{attribute 'linkalways'} 
{attribute 'no_explicit_call' := 'This FB is a CLASS and must be accessed using methods or properties'}
{attribute 'enable_dynamic_creation'}
FUNCTION_BLOCK AsynchronousRpcHandlers IMPLEMENTS I_AsynchronousRpcHandlers, I_HostAsynchronousRpcHandlers
VAR
	handlers : Dictionary;
	_hasHandlers : BOOL;
END_VAR

PROPERTY PUBLIC HasHandlers : BOOL
GET
HasHandlers := _hasHandlers;
END_GET
END_PROPERTY

METHOD PUBLIC RegisterHandler
VAR_INPUT
	MethodName : T_MAXSTRING;
	Handler : I_AsynchronousRpcHandler;
END_VAR
handlers.AddOrUpdate(MethodName, Handler);
_hasHandlers := true;
END_METHOD

METHOD PUBLIC TryGetByMethodName : BOOL
VAR_INPUT
	MethodName : T_MAXSTRING;
	Destination : REFERENCE TO I_AsynchronousRpcHandler;
END_VAR
TryGetByMethodName := handlers.TryGetValue(MethodName, Destination);
END_METHOD

END_FUNCTION_BLOCK

(* stored: Version 1.1.0.1, ProductVersion 3.1.4024.12
   POU AsynchronousRpcHandlers: Id {cd13ebd0-3788-4442-8ef7-64929a08abe4}, SpecialFunc None
   Property HasHandlers: Id {17926476-6420-47b5-979d-bcd741790e01}
   Get Get: Id {68a58ba0-9e12-4a74-b13d-27aec2ca21d2}
   Method RegisterHandler: Id {6a0cc49c-48db-4e06-80c7-262017cc9b6f}
   Method TryGetByMethodName: Id {22babab6-a3ca-4500-9900-ad0f417bd742} *)
